(*
Nazwa:			P05_Weight
Opis:			Stacja wagi
Wersja:			v0.2
Data:			2019-10-1
Autor:			DP
Urzadzenia:		
Konfiguracja:	
Info:
-przerobione na wagę beckhofa
*)
PROGRAM P05_Weight
VAR_INPUT
	IbWeight1FormSensor						AT %I*		: BOOL;							//Czujnik nad Waga 1
	IbWeight2FormSensor						AT %I*		: BOOL;							//Czujnik nad Waga 2
	IbWeight3FormSensor						AT %I*		: BOOL;							//Czujnik nad Waga 3
	IbWeight4FormSensor						AT %I*		: BOOL;							//Czujnik nad Waga 4
	IbWeight5FormSensor						AT %I*		: BOOL;							//Czujnik nad Waga 4
	IbWeight6FormSensor						AT %I*		: BOOL;							//Czujnik nad Waga 4
END_VAR
VAR
	//Podnosnik szalek
	
	//eWeightLiftRunningState			:E_WeightLiftState;				// Stan pracy podajnika
	fbWeightLiftState					:FB_State;
	
	//Waga 1
	fbWeight1							:FB_BeckhoffEL3356Weight;		// Blok sterujący pierwszą wagą
	eWeight1State						:E_Station; 					// Stan pracy podajnika platynek			
	eWeight1RunningState				:E_WeightState; 				// Stan pracy podajnika platynek
	fbWeight1State						:FB_State;					

	(*No nowej wagi*)
	(*wejścia*)
	InWeight1Value						 AT %I*: DINT;			// Wartość wagi
	IbWeight1Overrange					 AT %I*: BOOL;						
	IbWeight1DataInvalid				 AT %I*: BOOL;		
	IbWeight1Error 						 AT %I*: BOOL;	
	IbWeight1CalibrationInProgress 		 AT %I*: BOOL;
	IbWeight1SteadyState				 AT %I*: BOOL;
	IbWeight1SyncError 					 AT %I*: BOOL;
	(*wyjścia*)
	QbWeight1StartCalibration 			 AT %Q*: BOOL;
	QbWeight1DisableCalibration     	 AT %Q*: BOOL;
	QbWeight1InputFreeze 				 AT %Q*: BOOL;
	QbWeight1SampleMode 				 AT %Q*: BOOL;
	QbWeight1Tara 					     AT %Q*: BOOL;
	
	(*Ostrzezenia*)
	bWeight1Warning1					:BOOL; // 
	tonWeight1Tare						:TON;
	
	//Waga 2
	fbWeight2							:FB_BeckhoffEL3356Weight;		// Blok sterujący pierwszą wagą
	eWeight2State						:E_Station; 					// Stan pracy podajnika platynek			
	eWeight2RunningState				:E_WeightState; 				// Stan pracy podajnika platynek
	fbWeight2State						:FB_State;					

	(*No nowej wagi*)
	(*wejścia*)
	InWeight2Value 						AT %I*: DINT;			// Wartość wagi
	IbWeight2Overrange 					AT %I*: BOOL;						
	IbWeight2DataInvalid 				AT %I*: BOOL;		
	IbWeight2Error 						AT %I*: BOOL;	
	IbWeight2CalibrationInProgress		AT %I*: BOOL;
	IbWeight2SteadyState 				AT %I*: BOOL;
	IbWeight2SyncError 					AT %I*: BOOL;
	(*wyjścia*)
	QbWeight2StartCalibration 			AT %Q*: BOOL;
	QbWeight2DisableCalibration			AT %Q*: BOOL;
	QbWeight2InputFreeze 				AT %Q*: BOOL;
	QbWeight2SampleMode 				AT %Q*: BOOL;
	QbWeight2Tara 						AT %Q*: BOOL;
	
	(*Ostrzezenia*)
	bWeight2Warning1					:BOOL; // 
	tonWeight2Tare						:TON;
		
	//Waga 3
	fbWeight3							:FB_BeckhoffEL3356Weight;		// Blok sterujący pierwszą wagą
	eWeight3State						:E_Station; 					// Stan pracy podajnika platynek			
	eWeight3RunningState				:E_WeightState; 				// Stan pracy podajnika platynek
	fbWeight3State						:FB_State;					

	(*No nowej wagi*)
	(*wejścia*)
	InWeight3Value						 AT %I*: DINT;			// Wartość wagi
	IbWeight3Overrange 					 AT %I*: BOOL;						
	IbWeight3DataInvalid 				 AT %I*: BOOL;		
	IbWeight3Error 						 AT %I*: BOOL;	
	IbWeight3CalibrationInProgress 		 AT %I*: BOOL;
	IbWeight3SteadyState 				 AT %I*: BOOL;
	IbWeight3SyncError 					 AT %I*: BOOL;
	(*wyjścia*)
	QbWeight3StartCalibration 			 AT %Q*: BOOL;
	QbWeight3DisableCalibration 		 AT %Q*: BOOL;
	QbWeight3InputFreeze 				 AT %Q*: BOOL;
	QbWeight3SampleMode 			   	 AT %Q*: BOOL;
	QbWeight3Tara 						 AT %Q*: BOOL;
	
	(*Ostrzezenia*)
	bWeight3Warning1					:BOOL; // 
	tonWeight3Tare						: TON;	
	
	//Waga 4
	fbWeight4							:FB_BeckhoffEL3356Weight;		// Blok sterujący pierwszą wagą
	eWeight4State						:E_Station; 					// Stan pracy podajnika platynek			
	eWeight4RunningState				:E_WeightState; 				// Stan pracy podajnika platynek
	fbWeight4State						:FB_State;					

	(*No nowej wagi*)
	(*wejścia*)
	InWeight4Value 						AT %I*: DINT;			// Wartość wagi
	IbWeight4Overrange 					AT %I*: BOOL;						
	IbWeight4DataInvalid				AT %I*: BOOL;		
	IbWeight4Error 						AT %I*: BOOL;	
	IbWeight4CalibrationInProgress 		AT %I*: BOOL;
	IbWeight4SteadyState 				AT %I*: BOOL;
	IbWeight4SyncError 					AT %I*: BOOL;
	(*wyjścia*)
	QbWeight4StartCalibration 			AT %Q*: BOOL;
	QbWeight4DisableCalibration 		AT %Q*: BOOL;
	QbWeight4InputFreeze 				AT %Q*: BOOL;
	QbWeight4SampleMode 				AT %Q*: BOOL;
	QbWeight4Tara 						AT %Q*: BOOL;

	(*Ostrzezenia*)
	bWeight4Warning1					:BOOL; // 
	tonWeight4Tare						:TON;	
		
(******** Dozowanie dwufazowe******)	
////// Wagi przy dozowaniu dwufazowym dodano 07.04.2022
	//Waga 5
	fbWeight5							:FB_BeckhoffEL3356Weight;		// Blok sterujący pierwszą wagą
	eWeight5State						:E_Station; 					// Stan pracy podajnika platynek			
	eWeight5RunningState				:E_WeightState; 				// Stan pracy podajnika platynek
	fbWeight5State						:FB_State;					

	(*No nowej wagi*)
	(*wejścia*)
	InWeight5Value 						AT %I*: DINT;			// Wartość wagi
	IbWeight5Overrange 					AT %I*: BOOL;						
	IbWeight5DataInvalid 				AT %I*: BOOL;		
	IbWeight5Error 						AT %I*: BOOL;	
	IbWeight5CalibrationInProgress 		AT %I*: BOOL;
	IbWeight5SteadyState 				AT %I*: BOOL;
	IbWeight5SyncError 					AT %I*: BOOL;
	(*wyjścia*)
	QbWeight5StartCalibration 			AT %Q*: BOOL;
	QbWeight5DisableCalibration 		AT %Q*: BOOL;
	QbWeight5InputFreeze 				AT %Q*: BOOL;
	QbWeight5SampleMode 				AT %Q*: BOOL;
	QbWeight5Tara 						AT %Q*: BOOL;

	(*Ostrzezenia*)
	bWeight5Warning1					:BOOL; // 
	tonWeight5Tare						:TON;		
	
	//Waga 5
	fbWeight6							:FB_BeckhoffEL3356Weight;		// Blok sterujący pierwszą wagą
	eWeight6State						:E_Station; 					// Stan pracy podajnika platynek			
	eWeight6RunningState				:E_WeightState; 				// Stan pracy podajnika platynek
	fbWeight6State						:FB_State;					

	(*No nowej wagi*)
	(*wejścia*)
	InWeight6Value 						AT %I*: DINT;			// Wartość wagi
	IbWeight6Overrange 					AT %I*: BOOL;						
	IbWeight6DataInvalid 				AT %I*: BOOL;		
	IbWeight6Error 						AT %I*: BOOL;	
	IbWeight6CalibrationInProgress 		AT %I*: BOOL;
	IbWeight6SteadyState 				AT %I*: BOOL;
	IbWeight6SyncError 					AT %I*: BOOL;
	(*wyjścia*)
	QbWeight6StartCalibration 			AT %Q*: BOOL;
	QbWeight6DisableCalibration 		AT %Q*: BOOL;
	QbWeight6InputFreeze 				AT %Q*: BOOL;
	QbWeight6SampleMode 				AT %Q*: BOOL;
	QbWeight6Tara 						AT %Q*: BOOL;

	(*Ostrzezenia*)
	bWeight6Warning1					:BOOL; // 
	tonWeight6Tare						:TON;		
	
(******** Dozowanie dwufazowe******)		
	
	//Czujniki optyczne przed i za wagą
	fbFilterWeight1: FB_FilterEx;
	fbFilterWeight2: FB_FilterEx;
	fbFilterWeight3: FB_FilterEx;
	fbFilterWeight4: FB_FilterEx;
	fbFilterWeight5: FB_FilterEx;(****** dodane 07.04.2022 przy dodzowniu dwufazowym	**)
	fbFilterWeight6: FB_FilterEx;(****** dodane 07.04.2022 przy dodzowniu dwufazowym	**)

	rFilteredWeight1Value: REAL;
	rFilteredWeight2Value: REAL;
	rFilteredWeight3Value: REAL;
	rFilteredWeight4Value: REAL;
	rFilteredWeight5Value: REAL;(****** dodane 07.04.2022 przy dodzowniu dwufazowym	**)
	rFilteredWeight6Value: REAL;(****** dodane 07.04.2022 przy dodzowniu dwufazowym	**)
	
	//Damian dodane 2 fazy
	fbWeightStation2Phase							: FB_WeightStation;	
	eWeightStation2PhaseState						: E_Station;
	eWeightStation2PhaseRunningState				: E_WeightLiftStationState;
	
	//Dodane Przez Mikołaja
	fbWeightStation									: FB_WeightStation;
	eWeightStationState								: E_Station;
	eWeightStationRunningState						: E_WeightLiftStationState;
	
	IbWeight1ActuatorSensorUp			AT %I*		: BOOL;							//Czujnik podnoszenia Waga 1
	IbWeight2ActuatorSensorUp			AT %I*		: BOOL;							//Czujnik podnoszenia Waga 2
	IbWeight3ActuatorSensorUp			AT %I*		: BOOL;							//Czujnik podnoszenia Waga 3
	IbWeight4ActuatorSensorUp			AT %I*		: BOOL;							//Czujnik podnoszenia Waga 4
	IbWeight5ActuatorSensorUp			AT %I*		: BOOL;							//Czujnik podnoszenia Waga 5 
	IbWeight6ActuatorSensorUp			AT %I*		: BOOL;							//Czujnik podnoszenia Waga 6 
		
	QbWeight1Actuator								: BOOL;							//Podnoszenie Waga 1
    QbWeight2Actuator								: BOOL;							//Podnoszenie Waga 2
	QbWeight3Actuator								: BOOL;							//Podnoszenie Waga 3
	QbWeight4Actuator								: BOOL;							//Podnoszenie Waga 4	                                    		
	QbWeight5Actuator								: BOOL;							//Podnoszenie Waga 5 (2faza)	                                    		
	QbWeight6Actuator								: BOOL;							//Podnoszenie Waga 6 (2faza)

		
	(*Symulacja czujników*)
	tonIbWeight1ActuatorSensorUp					: TON;	
	tonIbWeight2ActuatorSensorUp					: TON;	
	tonIbWeight3ActuatorSensorUp					: TON;	
	tonIbWeight4ActuatorSensorUp					: TON;	
	tonIbWeight5ActuatorSensorUp					: TON;	
	tonIbWeight6ActuatorSensorUp					: TON;	
	
	tonIbWeight1FormSensor: TON;
	tonIbWeight2FormSensor: TON;
	tonIbWeight3FormSensor: TON;
	tonIbWeight4FormSensor: TON;
	tonIbWeight5FormSensor: TON;
	tonIbWeight6FormSensor: TON;
	
	fbIbWeight1FormBeforeSensor: FB_InputFilter_v2;
	fbIbWeight2FormBeforeSensor: FB_InputFilter_v2;
	fbIbWeight3FormBeforeSensor: FB_InputFilter_v2;
	fbIbWeight4FormBeforeSensor: FB_InputFilter_v2;		
	fbIbWeight5FormBeforeSensor: FB_InputFilter_v2;		
	fbIbWeight6FormBeforeSensor: FB_InputFilter_v2;			
	btemp: BOOL;
	
	//wykresy
	fbTrig1 : R_TRIG;
    fbTrig2 : R_TRIG;
    fbTrig3 : R_TRIG;
    fbTrig4 : R_TRIG;
	tSys : DT;
    tTOD : TOD;
	GetTimeSeconds : INT;
	weightIndex : INT;   // 0..7
    valueY : INT;
	i : INT;
	 
	fbHistory: FB_WeightHistory;
END_VAR


fbWeight1.bIgnoreError:=fbWeight2.bIgnoreError:=fbWeight3.bIgnoreError:=fbWeight4.bIgnoreError:=fbWeight5.bIgnoreError:=fbWeight6.bIgnoreError;

aFilter();
aWeight1();
aWeight2();
aWeight3();
aWeight4();
aWeight5();
aWeight6();
ACT_WeightChartDrawers();
IF NOT bDosingTwoPhases THEN
	ACT_WeightStation();
ELSE
	ACT_WeightStation2Phase();
END_IF

// Czas opóżnienia zbierania próbekFB_EntranceGatesServo
fbWeight1.nWeightingDelay:=fbWeight2.nWeightingDelay:=fbWeight3.nWeightingDelay:=fbWeight4.nWeightingDelay:=530;//530
fbWeight5.nWeightingDelay:=fbWeight6.nWeightingDelay:=750;//było 685

(********* GENEROWANIE STANU STACJI DO WIZKI**********)

fbWeight1State(
	eState															:= eWeight1State , 
	bRun															:= VIS.bWeight1DoWeighting,	
	eWeightRunningState												:= eWeight1RunningState , 
	sStateDesc														=> VIS.sWeight1State,
	iState															=> VIS.iWeight1State	);	

fbWeight2State(
	eState															:= eWeight2State , 
	bRun															:= VIS.bWeight2DoWeighting,	
	eWeightRunningState												:= eWeight2RunningState , 
	sStateDesc														=> VIS.sWeight2State,
	iState															=> VIS.iWeight2State	);	
		
fbWeight3State(
	eState															:= eWeight3State , 
	bRun															:= VIS.bWeight3DoWeighting,	
	eWeightRunningState												:= eWeight3RunningState , 
	sStateDesc														=> VIS.sWeight3State,
	iState															=> VIS.iWeight3State	);	
	
fbWeight4State(
	eState															:= eWeight4State , 
	bRun															:= VIS.bWeight4DoWeighting,	
	eWeightRunningState												:= eWeight4RunningState , 
	sStateDesc														=> VIS.sWeight4State,
	iState															=> VIS.iWeight4State	);	
	
fbWeight5State(
	eState															:= eWeight5State , 
	bRun															:= VIS.bWeight5DoWeighting,	
	eWeightRunningState												:= eWeight5RunningState , 
	sStateDesc														=> VIS.sWeight5State,
	iState															=> VIS.iWeight5State	);	

fbWeight6State(
	eState															:= eWeight6State , 
	bRun															:= VIS.bWeight6DoWeighting,	
	eWeightRunningState												:= eWeight6RunningState , 
	sStateDesc														=> VIS.sWeight6State,
	iState															=> VIS.iWeight6State	);		
	
fbWeightLiftState(
	eState															:= eWeightStationState, 
	bRun															:= VIS.bWeightLiftRun OR bWeightLift2PhaseRun,	
	eWeightLiftRunningState											:= eWeightStationRunningState , 
	sStateDesc														=> VIS.sWeightLiftState,
	iState															=> VIS.iWeightLiftState	);		
	
(***** KONIEC GENEROWANIE STANU STACJI DO WIZKI*******)

(****Ostrzezenia***)
// Waga 1
WeightWarning[0].sDescription										:= 'Wagi | Brak stabilizacji przy pomiarach';
IF (bWeight1Warning1 OR bWeight2Warning1 OR bWeight3Warning1 OR bWeight4Warning1 OR bWeight5Warning1 OR bWeight6Warning1) AND NOT WeightWarning[0].bWarning THEN
	WeightWarning[0].bWarning										:= TRUE;
	
ELSIF NOT bWeight1Warning1 AND WeightWarning[0].bAcknowledge THEN
	WeightWarning[0].bWarning										:= FALSE;
	WeightWarning[0].bAcknowledge									:= FALSE;
	VIS.uliWarningAcknowledge.4 										:= FALSE;
	
ELSIF WeightWarning[0].bAcknowledge THEN
	WeightWarning[0].bAcknowledge									:= TRUE;
END_IF


(********KASOWANIE ROZKAZÓW CYKLI*********)
IF fbWeight1.bCycleDone AND bManualMode THEN
	VIS.bWeight1DoWeighting 												:= FALSE;
END_IF

tonWeight1Tare(IN:=VIS.bWeight1Tare,PT:=T#2S);
IF tonWeight1Tare.Q THEN
	VIS.bWeight1Tare												:= FALSE;
END_IF

IF fbWeight2.bCycleDone AND bManualMode THEN
	VIS.bWeight2DoWeighting 												:= FALSE;
END_IF

tonWeight2Tare(IN:=VIS.bWeight2Tare,PT:=T#2S);
IF tonWeight2Tare.Q THEN
	VIS.bWeight2Tare												:= FALSE;
END_IF

IF fbWeight3.bCycleDone AND bManualMode THEN
	VIS.bWeight3DoWeighting 												:= FALSE;
END_IF

tonWeight3Tare(IN:=VIS.bWeight3Tare,PT:=T#2S);
IF tonWeight3Tare.Q THEN
	VIS.bWeight3Tare												:= FALSE;
END_IF
//
IF fbWeight4.bCycleDone AND bManualMode THEN
	VIS.bWeight4DoWeighting 												:= FALSE;
END_IF

tonWeight4Tare(IN:=VIS.bWeight4Tare,PT:=T#2S);
IF tonWeight4Tare.Q THEN
	VIS.bWeight4Tare												:= FALSE;
END_IF

// Waga 5 (1 stacja przy dwufazie)
IF fbWeight5.bCycleDone AND bManualMode THEN
	VIS.bWeight5DoWeighting 												:= FALSE;
END_IF

tonWeight5Tare(IN:=VIS.bWeight5Tare,PT:=T#2S);
IF tonWeight5Tare.Q THEN
	VIS.bWeight5Tare												:= FALSE;
END_IF

// Waga 6 (1 stacja przy dwufazie)
IF fbWeight6.bCycleDone AND bManualMode THEN
	VIS.bWeight6DoWeighting 												:= FALSE;
END_IF

tonWeight6Tare(IN:=VIS.bWeight6Tare,PT:=T#2S);
IF tonWeight6Tare.Q THEN
	VIS.bWeight6Tare												:= FALSE;
END_IF
(*****KONIEC KASOWANIA ROZKAZÓW CYKLI*****)

(**SYMULACJA CZUJNIKÓW**)
tonIbWeight1ActuatorSensorUp(IN:= QbWeight1Actuator, PT:=T#80MS);
tonIbWeight2ActuatorSensorUp(IN:= QbWeight2Actuator, PT:=T#80MS);
tonIbWeight3ActuatorSensorUp(IN:= QbWeight3Actuator, PT:=T#80MS);
tonIbWeight4ActuatorSensorUp(IN:= QbWeight4Actuator, PT:=T#80MS);
tonIbWeight5ActuatorSensorUp(IN:= QbWeight5Actuator, PT:=T#100MS);
tonIbWeight6ActuatorSensorUp(IN:= QbWeight6Actuator, PT:=T#100MS);

ACTION ACT_WeightChartDrawers:
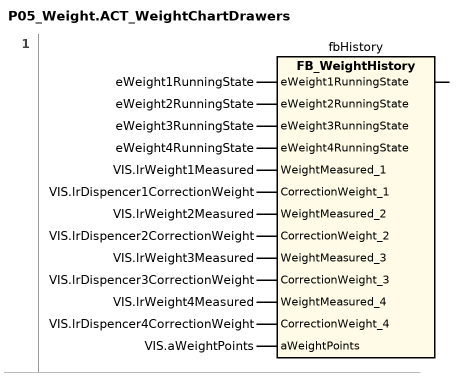
// NETWORK 1
fbHistory(
    eWeight1RunningState := eWeight1RunningState,
    eWeight2RunningState := eWeight2RunningState,
    eWeight3RunningState := eWeight3RunningState,
    eWeight4RunningState := eWeight4RunningState,
    WeightMeasured_1 := VIS.lrWeight1Measured,
    CorrectionWeight_1 := VIS.lrDispencer1CorrectionWeight,
    WeightMeasured_2 := VIS.lrWeight2Measured,
    CorrectionWeight_2 := VIS.lrDispencer2CorrectionWeight,
    WeightMeasured_3 := VIS.lrWeight3Measured,
    CorrectionWeight_3 := VIS.lrDispencer3CorrectionWeight,
    WeightMeasured_4 := VIS.lrWeight4Measured,
    CorrectionWeight_4 := VIS.lrDispencer4CorrectionWeight,
    aWeightPoints := VIS.aWeightPoints); // FB_WeightHistory
END_ACTION

ACTION ACT_WeightStation:
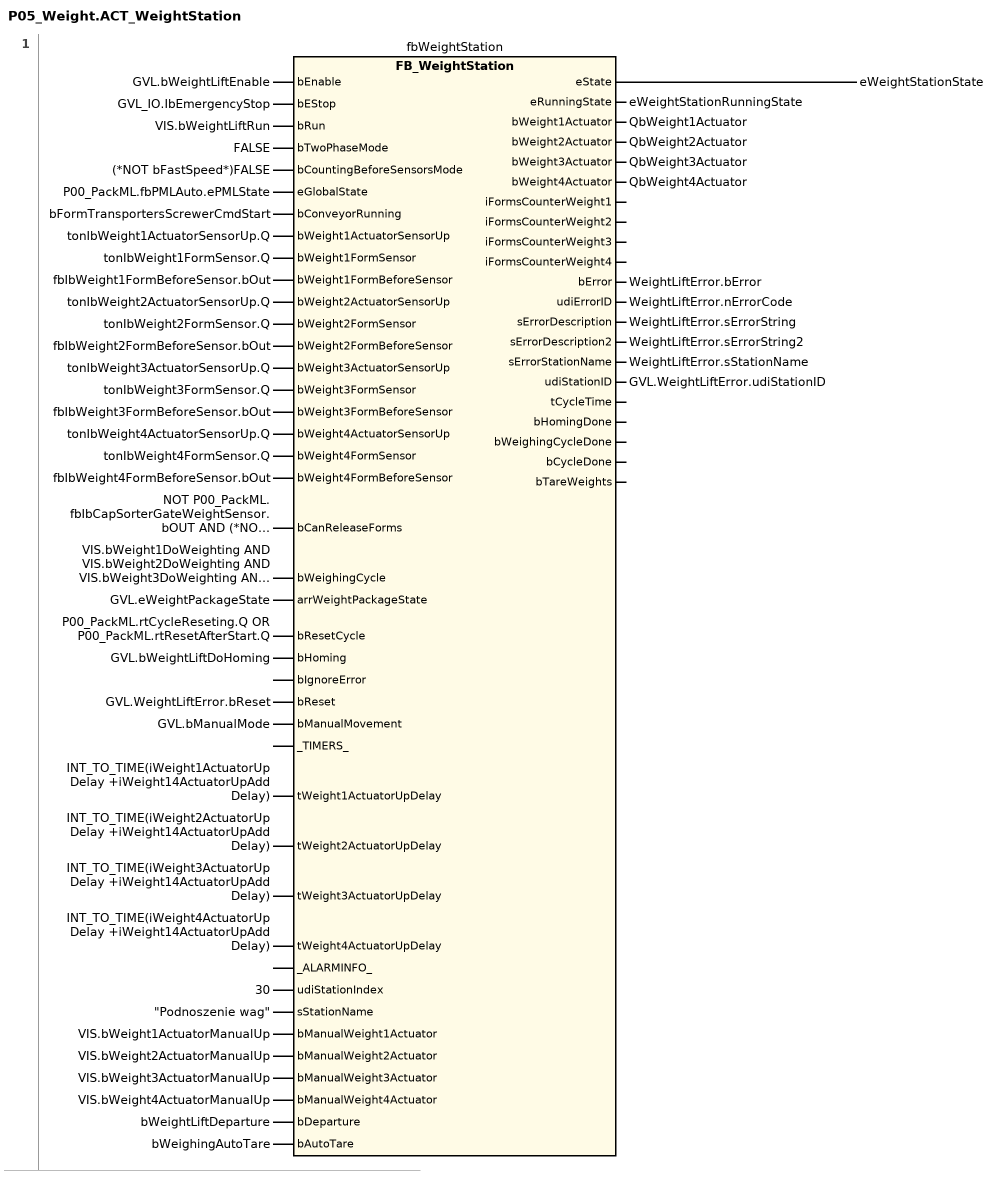
// NETWORK 1
fbWeightStation(
    bEnable := GVL.bWeightLiftEnable,
    bEStop := GVL_IO.IbEmergencyStop,
    bRun := VIS.bWeightLiftRun,
    bTwoPhaseMode := FALSE,
    bCountingBeforeSensorsMode := (*NOT bFastSpeed*)FALSE,
    eGlobalState := P00_PackML.fbPMLAuto.ePMLState,
    bConveyorRunning := bFormTransportersScrewerCmdStart,
    bWeight1ActuatorSensorUp := tonIbWeight1ActuatorSensorUp.Q,
    bWeight1FormSensor := tonIbWeight1FormSensor.Q,
    bWeight1FormBeforeSensor := fbIbWeight1FormBeforeSensor.bOut,
    bWeight2ActuatorSensorUp := tonIbWeight2ActuatorSensorUp.Q,
    bWeight2FormSensor := tonIbWeight2FormSensor.Q,
    bWeight2FormBeforeSensor := fbIbWeight2FormBeforeSensor.bOut,
    bWeight3ActuatorSensorUp := tonIbWeight3ActuatorSensorUp.Q,
    bWeight3FormSensor := tonIbWeight3FormSensor.Q,
    bWeight3FormBeforeSensor := fbIbWeight3FormBeforeSensor.bOut,
    bWeight4ActuatorSensorUp := tonIbWeight4ActuatorSensorUp.Q,
    bWeight4FormSensor := tonIbWeight4FormSensor.Q,
    bWeight4FormBeforeSensor := fbIbWeight4FormBeforeSensor.bOut,
    bCanReleaseForms := NOT P00_PackML.fbIbCapSorterGateWeightSensor.bOUT AND (*NOT P00_PackML.fbIbCapCorrectCheckFormSensor.bOUT AND zalezy od ilosci formatek*)  NOT bWeight1234ReleaseBlock,
    bWeighingCycle := VIS.bWeight1DoWeighting AND VIS.bWeight2DoWeighting AND VIS.bWeight3DoWeighting AND VIS.bWeight4DoWeighting,
    arrWeightPackageState := GVL.eWeightPackageState,
    bResetCycle := P00_PackML.rtCycleReseting.Q OR P00_PackML.rtResetAfterStart.Q,
    bHoming := GVL.bWeightLiftDoHoming,
    bReset := GVL.WeightLiftError.bReset,
    bManualMovement := GVL.bManualMode,
    tWeight1ActuatorUpDelay := INT_TO_TIME(iWeight1ActuatorUpDelay +iWeight14ActuatorUpAddDelay),
    tWeight2ActuatorUpDelay := INT_TO_TIME(iWeight2ActuatorUpDelay +iWeight14ActuatorUpAddDelay),
    tWeight3ActuatorUpDelay := INT_TO_TIME(iWeight3ActuatorUpDelay +iWeight14ActuatorUpAddDelay),
    tWeight4ActuatorUpDelay := INT_TO_TIME(iWeight4ActuatorUpDelay +iWeight14ActuatorUpAddDelay),
    udiStationIndex := 30,
    sStationName := "Podnoszenie wag",
    bManualWeight1Actuator := VIS.bWeight1ActuatorManualUp,
    bManualWeight2Actuator := VIS.bWeight2ActuatorManualUp,
    bManualWeight3Actuator := VIS.bWeight3ActuatorManualUp,
    bManualWeight4Actuator := VIS.bWeight4ActuatorManualUp,
    bDeparture := bWeightLiftDeparture,
    bAutoTare := bWeighingAutoTare,
    eRunningState => eWeightStationRunningState,
    bWeight1Actuator => QbWeight1Actuator,
    bWeight2Actuator => QbWeight2Actuator,
    bWeight3Actuator => QbWeight3Actuator,
    bWeight4Actuator => QbWeight4Actuator,
    bError => WeightLiftError.bError,
    udiErrorID => WeightLiftError.nErrorCode,
    sErrorDescription => WeightLiftError.sErrorString,
    sErrorDescription2 => WeightLiftError.sErrorString2,
    sErrorStationName => WeightLiftError.sStationName,
    udiStationID => GVL.WeightLiftError.udiStationID); // FB_WeightStation
eWeightStationState := fbWeightStation.eState;
END_ACTION

ACTION ACT_WeightStation2Phase:
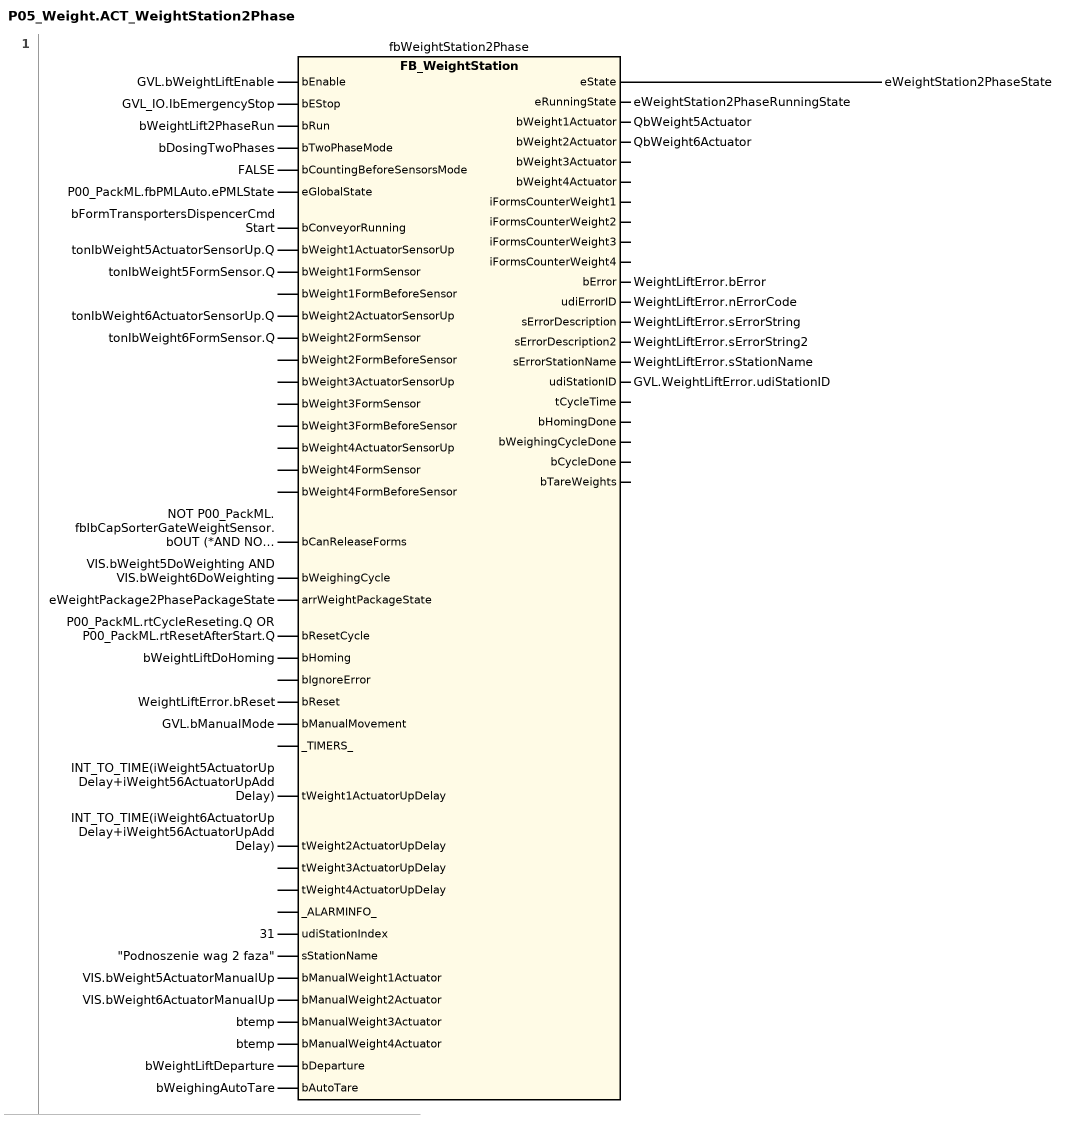
// NETWORK 1
fbWeightStation2Phase(
    bEnable := GVL.bWeightLiftEnable,
    bEStop := GVL_IO.IbEmergencyStop,
    bRun := bWeightLift2PhaseRun,
    bTwoPhaseMode := bDosingTwoPhases,
    bCountingBeforeSensorsMode := FALSE,
    eGlobalState := P00_PackML.fbPMLAuto.ePMLState,
    bConveyorRunning := bFormTransportersDispencerCmdStart,
    bWeight1ActuatorSensorUp := tonIbWeight5ActuatorSensorUp.Q,
    bWeight1FormSensor := tonIbWeight5FormSensor.Q,
    bWeight2ActuatorSensorUp := tonIbWeight6ActuatorSensorUp.Q,
    bWeight2FormSensor := tonIbWeight6FormSensor.Q,
    bCanReleaseForms := NOT P00_PackML.fbIbCapSorterGateWeightSensor.bOUT (*AND NOT P00_PackML.fbIbCapCorrectCheckFormSensor.bOUT*)  AND NOT bWeight56ReleaseBlock,
    bWeighingCycle := VIS.bWeight5DoWeighting AND VIS.bWeight6DoWeighting,
    arrWeightPackageState := eWeightPackage2PhasePackageState,
    bResetCycle := P00_PackML.rtCycleReseting.Q OR P00_PackML.rtResetAfterStart.Q,
    bHoming := bWeightLiftDoHoming,
    bReset := WeightLiftError.bReset,
    bManualMovement := GVL.bManualMode,
    tWeight1ActuatorUpDelay := INT_TO_TIME(iWeight5ActuatorUpDelay+iWeight56ActuatorUpAddDelay),
    tWeight2ActuatorUpDelay := INT_TO_TIME(iWeight6ActuatorUpDelay+iWeight56ActuatorUpAddDelay),
    udiStationIndex := 31,
    sStationName := "Podnoszenie wag 2 faza",
    bManualWeight1Actuator := VIS.bWeight5ActuatorManualUp,
    bManualWeight2Actuator := VIS.bWeight6ActuatorManualUp,
    bManualWeight3Actuator := btemp,
    bManualWeight4Actuator := btemp,
    bDeparture := bWeightLiftDeparture,
    bAutoTare := bWeighingAutoTare,
    eRunningState => eWeightStation2PhaseRunningState,
    bWeight1Actuator => QbWeight5Actuator,
    bWeight2Actuator => QbWeight6Actuator,
    bError => WeightLiftError.bError,
    udiErrorID => WeightLiftError.nErrorCode,
    sErrorDescription => WeightLiftError.sErrorString,
    sErrorDescription2 => WeightLiftError.sErrorString2,
    sErrorStationName => WeightLiftError.sStationName,
    udiStationID => GVL.WeightLiftError.udiStationID); // FB_WeightStation
eWeightStation2PhaseState := fbWeightStation2Phase.eState;
END_ACTION

ACTION aFilter:
fbFilterWeight1(
				rIn:=				DINT_TO_REAL(InWeight1Value), 
				tTimeConstant:= 	T#25MS, //bylo 25
				rOut=>				rFilteredWeight1Value);
							
fbFilterWeight2(
				rIn:=				DINT_TO_REAL(InWeight2Value), 
				tTimeConstant:= 	T#25MS, //bylo 25
				rOut=>				rFilteredWeight2Value);
				
fbFilterWeight3(
				rIn:=				DINT_TO_REAL(InWeight3Value), 
				tTimeConstant:= 	T#52MS, //bylo 25
				rOut=>				rFilteredWeight3Value);
				
fbFilterWeight4(
				rIn:=				DINT_TO_REAL(InWeight4Value), 
				tTimeConstant:= 	T#25MS, //bylo 25
				rOut=>				rFilteredWeight4Value);
///////////////////////////////////////////////////////////////////////////////				
fbFilterWeight5(
				rIn:=				DINT_TO_REAL(InWeight5Value), 
				tTimeConstant:= 	T#25MS, //bylo 25
				rOut=>				rFilteredWeight5Value);
								
fbFilterWeight6(
				rIn:=				DINT_TO_REAL(InWeight6Value), 
				tTimeConstant:= 	T#25MS, //bylo 25
				rOut=>				rFilteredWeight6Value);														
/////////////////////////////////////////////////////////////////////////////

tonIbWeight1FormSensor			(IN:=IbWeight1FormSensor ,		PT:=T#120MS); //160
tonIbWeight2FormSensor			(IN:=IbWeight2FormSensor ,		PT:=T#120MS); //160
tonIbWeight3FormSensor			(IN:=IbWeight3FormSensor ,		PT:=T#120MS); //160
tonIbWeight4FormSensor			(IN:=IbWeight4FormSensor ,		PT:=T#120MS); //160
tonIbWeight5FormSensor			(IN:=IbWeight5FormSensor ,		PT:=T#120MS); //60
tonIbWeight6FormSensor			(IN:=IbWeight6FormSensor ,		PT:=T#120MS); //60

IF VIS.nFormTransportersScrewerVelocitySVShow < 500 THEN
	fbIbWeight1FormBeforeSensor	(bIN:=IbWeight1ActuatorSensorUp,	tFilterTimeOn:=T#70MS,	tFilterTimeOff:=T#150MS);
	fbIbWeight2FormBeforeSensor	(bIN:=IbWeight2ActuatorSensorUp,	tFilterTimeOn:=T#70MS,	tFilterTimeOff:=T#150MS);
	fbIbWeight3FormBeforeSensor	(bIN:=IbWeight3ActuatorSensorUp,	tFilterTimeOn:=T#70MS,	tFilterTimeOff:=T#150MS);
	fbIbWeight4FormBeforeSensor	(bIN:=IbWeight4ActuatorSensorUp,	tFilterTimeOn:=T#70MS,	tFilterTimeOff:=T#150MS);
ELSE
	fbIbWeight1FormBeforeSensor	(bIN:=IbWeight1ActuatorSensorUp,	tFilterTimeOn:=T#10MS,	tFilterTimeOff:=T#10MS);//bylo 40 i 20
	fbIbWeight2FormBeforeSensor	(bIN:=IbWeight2ActuatorSensorUp,	tFilterTimeOn:=T#10MS,	tFilterTimeOff:=T#10MS);//bylo 40 i 20
	fbIbWeight3FormBeforeSensor	(bIN:=IbWeight3ActuatorSensorUp,	tFilterTimeOn:=T#10MS,	tFilterTimeOff:=T#10MS);//bylo 40 i 20
	fbIbWeight4FormBeforeSensor	(bIN:=IbWeight4ActuatorSensorUp,	tFilterTimeOn:=T#10MS,	tFilterTimeOff:=T#10MS);//bylo 40 i 20	
END_IF

IF VIS.nFormTransportersDispencerVelocitySVShow < 500 THEN
	fbIbWeight5FormBeforeSensor	(bIN:=IbWeight5FormSensor,			tFilterTimeOn:=T#70MS,	tFilterTimeOff:=T#150MS);
	fbIbWeight6FormBeforeSensor	(bIN:=IbWeight6FormSensor,			tFilterTimeOn:=T#70MS,	tFilterTimeOff:=T#150MS);
ELSE
	fbIbWeight5FormBeforeSensor	(bIN:=IbWeight5FormSensor,			tFilterTimeOn:=T#70MS,	tFilterTimeOff:=T#150MS);
	fbIbWeight6FormBeforeSensor	(bIN:=IbWeight6FormSensor,			tFilterTimeOn:=T#70MS,	tFilterTimeOff:=T#150MS);
END_IF
END_ACTION

ACTION aWeight1:
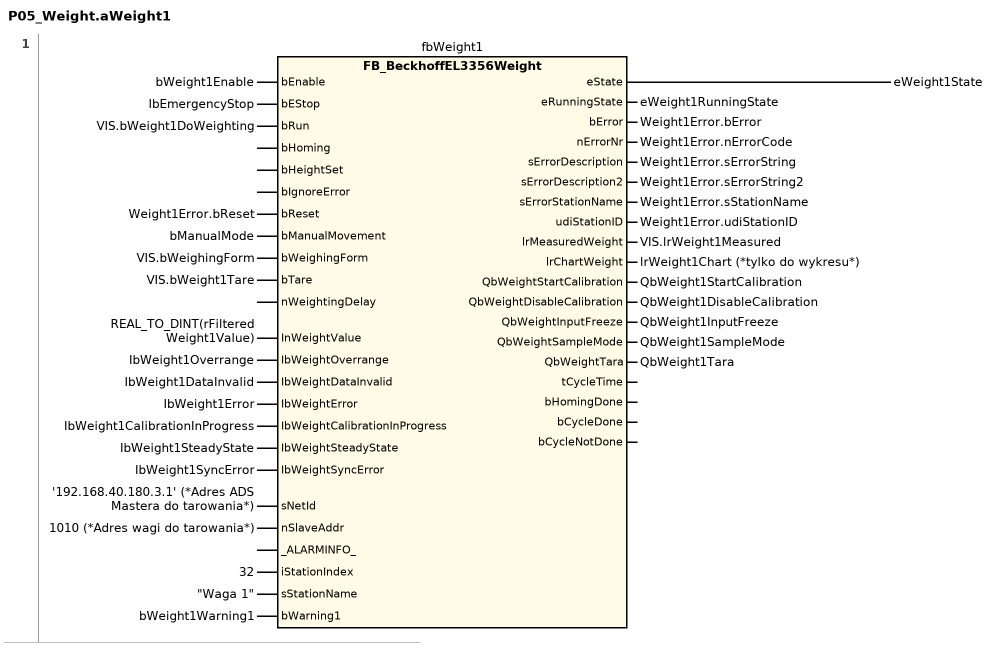
// NETWORK 1
fbWeight1(
    bEnable := bWeight1Enable,
    bEStop := IbEmergencyStop,
    bRun := VIS.bWeight1DoWeighting,
    bReset := Weight1Error.bReset,
    bManualMovement := bManualMode,
    bWeighingForm := VIS.bWeighingForm,
    bTare := VIS.bWeight1Tare,
    InWeightValue := REAL_TO_DINT(rFilteredWeight1Value),
    IbWeightOverrange := IbWeight1Overrange,
    IbWeightDataInvalid := IbWeight1DataInvalid,
    IbWeightError := IbWeight1Error,
    IbWeightCalibrationInProgress := IbWeight1CalibrationInProgress,
    IbWeightSteadyState := IbWeight1SteadyState,
    IbWeightSyncError := IbWeight1SyncError,
    sNetId := '192.168.40.180.3.1' (*Adres ADS Mastera do tarowania*),
    nSlaveAddr := 1010 (*Adres wagi do tarowania*),
    iStationIndex := 32,
    sStationName := "Waga 1",
    bWarning1 := bWeight1Warning1,
    eRunningState => eWeight1RunningState,
    bError => Weight1Error.bError,
    nErrorNr => Weight1Error.nErrorCode,
    sErrorDescription => Weight1Error.sErrorString,
    sErrorDescription2 => Weight1Error.sErrorString2,
    sErrorStationName => Weight1Error.sStationName,
    udiStationID => Weight1Error.udiStationID,
    lrMeasuredWeight => VIS.lrWeight1Measured,
    lrChartWeight => lrWeight1Chart (*tylko do wykresu*),
    QbWeightStartCalibration => QbWeight1StartCalibration,
    QbWeightDisableCalibration => QbWeight1DisableCalibration,
    QbWeightInputFreeze => QbWeight1InputFreeze,
    QbWeightSampleMode => QbWeight1SampleMode,
    QbWeightTara => QbWeight1Tara); // FB_BeckhoffEL3356Weight
eWeight1State := fbWeight1.eState;
END_ACTION

ACTION aWeight2:
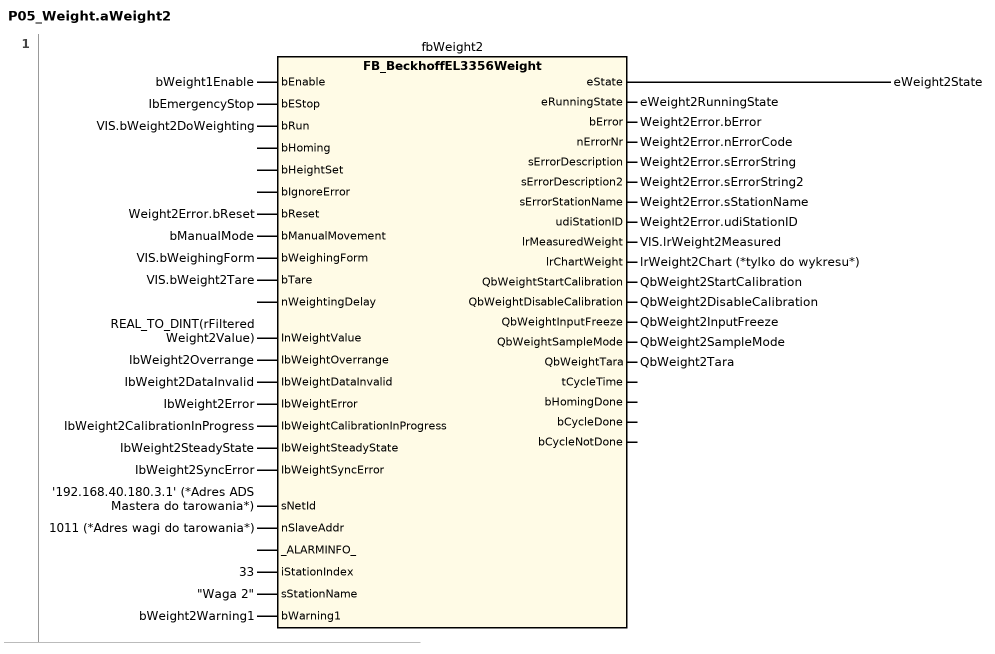
// NETWORK 1
fbWeight2(
    bEnable := bWeight1Enable,
    bEStop := IbEmergencyStop,
    bRun := VIS.bWeight2DoWeighting,
    bReset := Weight2Error.bReset,
    bManualMovement := bManualMode,
    bWeighingForm := VIS.bWeighingForm,
    bTare := VIS.bWeight2Tare,
    InWeightValue := REAL_TO_DINT(rFilteredWeight2Value),
    IbWeightOverrange := IbWeight2Overrange,
    IbWeightDataInvalid := IbWeight2DataInvalid,
    IbWeightError := IbWeight2Error,
    IbWeightCalibrationInProgress := IbWeight2CalibrationInProgress,
    IbWeightSteadyState := IbWeight2SteadyState,
    IbWeightSyncError := IbWeight2SyncError,
    sNetId := '192.168.40.180.3.1' (*Adres ADS Mastera do tarowania*),
    nSlaveAddr := 1011 (*Adres wagi do tarowania*),
    iStationIndex := 33,
    sStationName := "Waga 2",
    bWarning1 := bWeight2Warning1,
    eRunningState => eWeight2RunningState,
    bError => Weight2Error.bError,
    nErrorNr => Weight2Error.nErrorCode,
    sErrorDescription => Weight2Error.sErrorString,
    sErrorDescription2 => Weight2Error.sErrorString2,
    sErrorStationName => Weight2Error.sStationName,
    udiStationID => Weight2Error.udiStationID,
    lrMeasuredWeight => VIS.lrWeight2Measured,
    lrChartWeight => lrWeight2Chart (*tylko do wykresu*),
    QbWeightStartCalibration => QbWeight2StartCalibration,
    QbWeightDisableCalibration => QbWeight2DisableCalibration,
    QbWeightInputFreeze => QbWeight2InputFreeze,
    QbWeightSampleMode => QbWeight2SampleMode,
    QbWeightTara => QbWeight2Tara); // FB_BeckhoffEL3356Weight
eWeight2State := fbWeight2.eState;
END_ACTION

ACTION aWeight3:
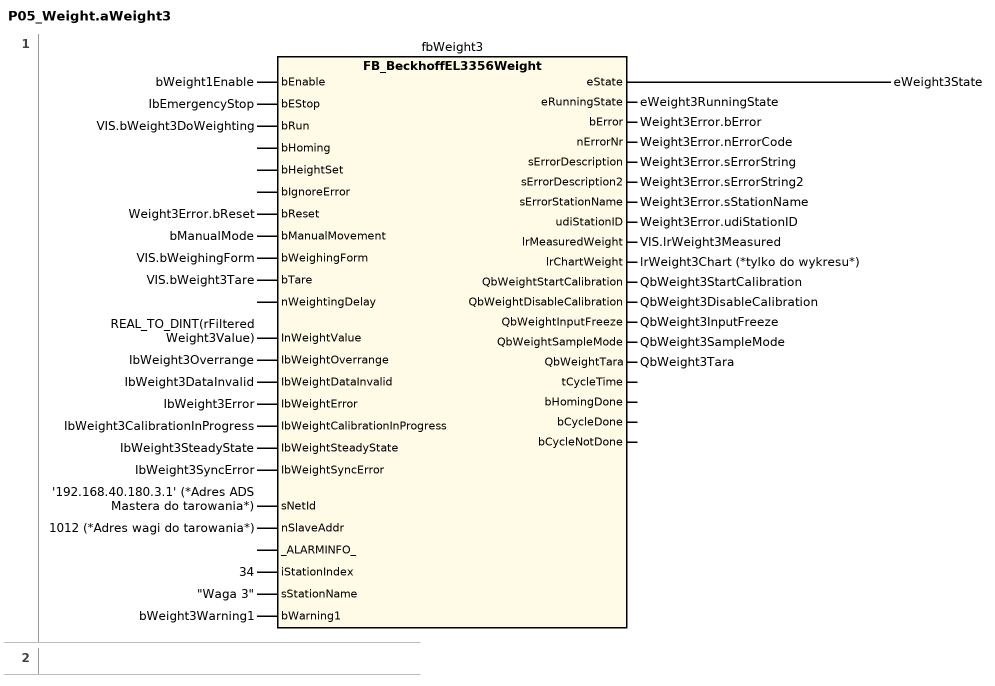
// NETWORK 1
fbWeight3(
    bEnable := bWeight1Enable,
    bEStop := IbEmergencyStop,
    bRun := VIS.bWeight3DoWeighting,
    bReset := Weight3Error.bReset,
    bManualMovement := bManualMode,
    bWeighingForm := VIS.bWeighingForm,
    bTare := VIS.bWeight3Tare,
    InWeightValue := REAL_TO_DINT(rFilteredWeight3Value),
    IbWeightOverrange := IbWeight3Overrange,
    IbWeightDataInvalid := IbWeight3DataInvalid,
    IbWeightError := IbWeight3Error,
    IbWeightCalibrationInProgress := IbWeight3CalibrationInProgress,
    IbWeightSteadyState := IbWeight3SteadyState,
    IbWeightSyncError := IbWeight3SyncError,
    sNetId := '192.168.40.180.3.1' (*Adres ADS Mastera do tarowania*),
    nSlaveAddr := 1012 (*Adres wagi do tarowania*),
    iStationIndex := 34,
    sStationName := "Waga 3",
    bWarning1 := bWeight3Warning1,
    eRunningState => eWeight3RunningState,
    bError => Weight3Error.bError,
    nErrorNr => Weight3Error.nErrorCode,
    sErrorDescription => Weight3Error.sErrorString,
    sErrorDescription2 => Weight3Error.sErrorString2,
    sErrorStationName => Weight3Error.sStationName,
    udiStationID => Weight3Error.udiStationID,
    lrMeasuredWeight => VIS.lrWeight3Measured,
    lrChartWeight => lrWeight3Chart (*tylko do wykresu*),
    QbWeightStartCalibration => QbWeight3StartCalibration,
    QbWeightDisableCalibration => QbWeight3DisableCalibration,
    QbWeightInputFreeze => QbWeight3InputFreeze,
    QbWeightSampleMode => QbWeight3SampleMode,
    QbWeightTara => QbWeight3Tara); // FB_BeckhoffEL3356Weight
eWeight3State := fbWeight3.eState;

// NETWORK 2
END_ACTION

ACTION aWeight4:
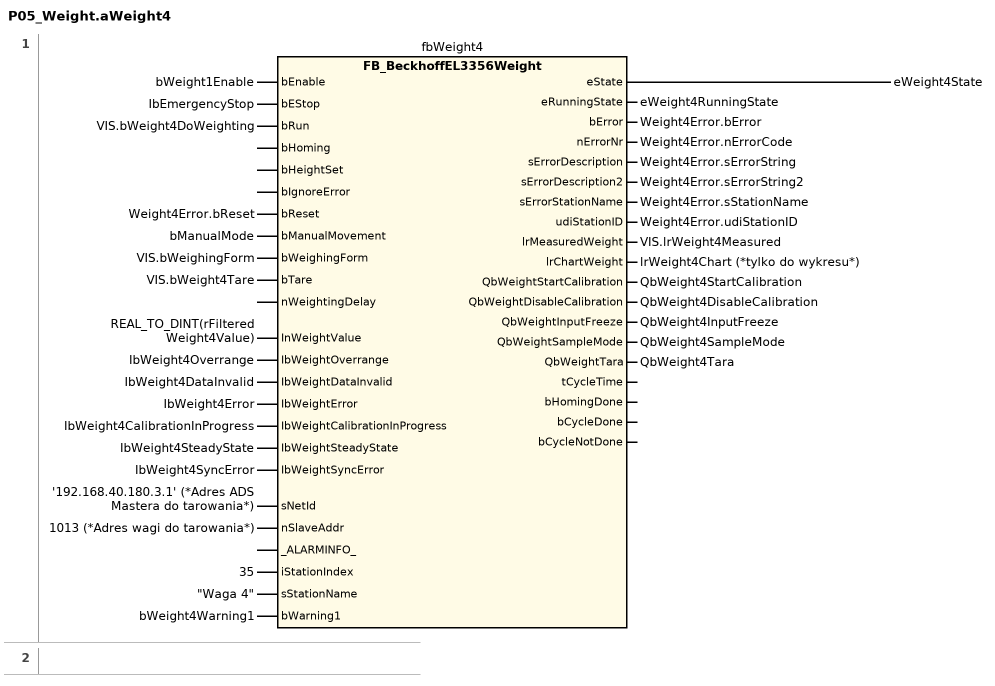
// NETWORK 1
fbWeight4(
    bEnable := bWeight1Enable,
    bEStop := IbEmergencyStop,
    bRun := VIS.bWeight4DoWeighting,
    bReset := Weight4Error.bReset,
    bManualMovement := bManualMode,
    bWeighingForm := VIS.bWeighingForm,
    bTare := VIS.bWeight4Tare,
    InWeightValue := REAL_TO_DINT(rFilteredWeight4Value),
    IbWeightOverrange := IbWeight4Overrange,
    IbWeightDataInvalid := IbWeight4DataInvalid,
    IbWeightError := IbWeight4Error,
    IbWeightCalibrationInProgress := IbWeight4CalibrationInProgress,
    IbWeightSteadyState := IbWeight4SteadyState,
    IbWeightSyncError := IbWeight4SyncError,
    sNetId := '192.168.40.180.3.1' (*Adres ADS Mastera do tarowania*),
    nSlaveAddr := 1013 (*Adres wagi do tarowania*),
    iStationIndex := 35,
    sStationName := "Waga 4",
    bWarning1 := bWeight4Warning1,
    eRunningState => eWeight4RunningState,
    bError => Weight4Error.bError,
    nErrorNr => Weight4Error.nErrorCode,
    sErrorDescription => Weight4Error.sErrorString,
    sErrorDescription2 => Weight4Error.sErrorString2,
    sErrorStationName => Weight4Error.sStationName,
    udiStationID => Weight4Error.udiStationID,
    lrMeasuredWeight => VIS.lrWeight4Measured,
    lrChartWeight => lrWeight4Chart (*tylko do wykresu*),
    QbWeightStartCalibration => QbWeight4StartCalibration,
    QbWeightDisableCalibration => QbWeight4DisableCalibration,
    QbWeightInputFreeze => QbWeight4InputFreeze,
    QbWeightSampleMode => QbWeight4SampleMode,
    QbWeightTara => QbWeight4Tara); // FB_BeckhoffEL3356Weight
eWeight4State := fbWeight4.eState;

// NETWORK 2
END_ACTION

ACTION aWeight5:
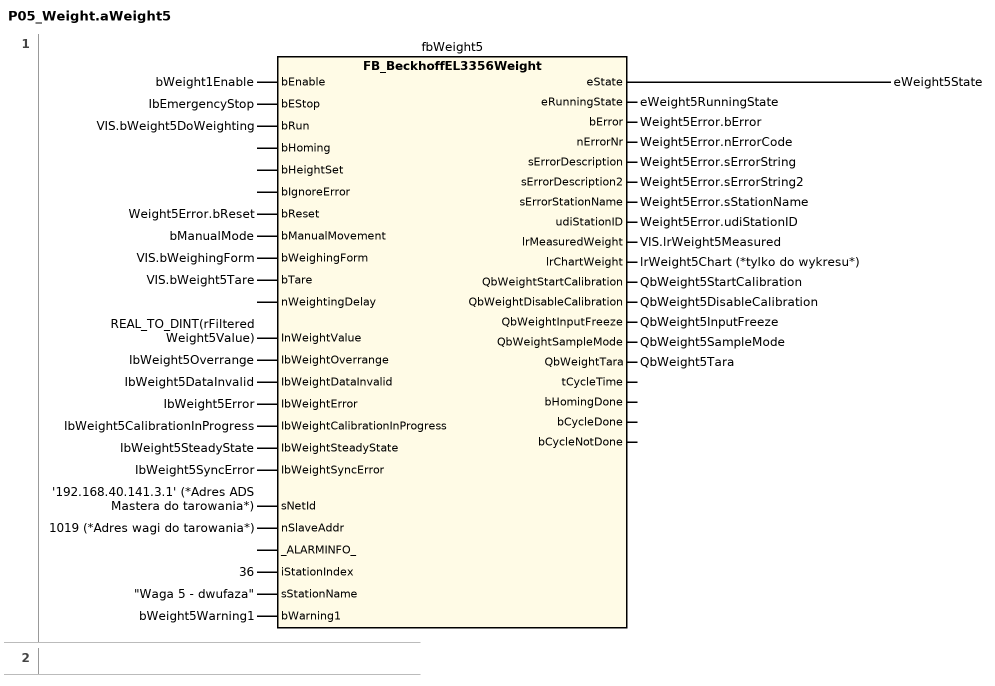
// NETWORK 1
fbWeight5(
    bEnable := bWeight1Enable,
    bEStop := IbEmergencyStop,
    bRun := VIS.bWeight5DoWeighting,
    bReset := Weight5Error.bReset,
    bManualMovement := bManualMode,
    bWeighingForm := VIS.bWeighingForm,
    bTare := VIS.bWeight5Tare,
    InWeightValue := REAL_TO_DINT(rFilteredWeight5Value),
    IbWeightOverrange := IbWeight5Overrange,
    IbWeightDataInvalid := IbWeight5DataInvalid,
    IbWeightError := IbWeight5Error,
    IbWeightCalibrationInProgress := IbWeight5CalibrationInProgress,
    IbWeightSteadyState := IbWeight5SteadyState,
    IbWeightSyncError := IbWeight5SyncError,
    sNetId := '192.168.40.141.3.1' (*Adres ADS Mastera do tarowania*),
    nSlaveAddr := 1019 (*Adres wagi do tarowania*),
    iStationIndex := 36,
    sStationName := "Waga 5 - dwufaza",
    bWarning1 := bWeight5Warning1,
    eRunningState => eWeight5RunningState,
    bError => Weight5Error.bError,
    nErrorNr => Weight5Error.nErrorCode,
    sErrorDescription => Weight5Error.sErrorString,
    sErrorDescription2 => Weight5Error.sErrorString2,
    sErrorStationName => Weight5Error.sStationName,
    udiStationID => Weight5Error.udiStationID,
    lrMeasuredWeight => VIS.lrWeight5Measured,
    lrChartWeight => lrWeight5Chart (*tylko do wykresu*),
    QbWeightStartCalibration => QbWeight5StartCalibration,
    QbWeightDisableCalibration => QbWeight5DisableCalibration,
    QbWeightInputFreeze => QbWeight5InputFreeze,
    QbWeightSampleMode => QbWeight5SampleMode,
    QbWeightTara => QbWeight5Tara); // FB_BeckhoffEL3356Weight
eWeight5State := fbWeight5.eState;

// NETWORK 2
END_ACTION

ACTION aWeight6:
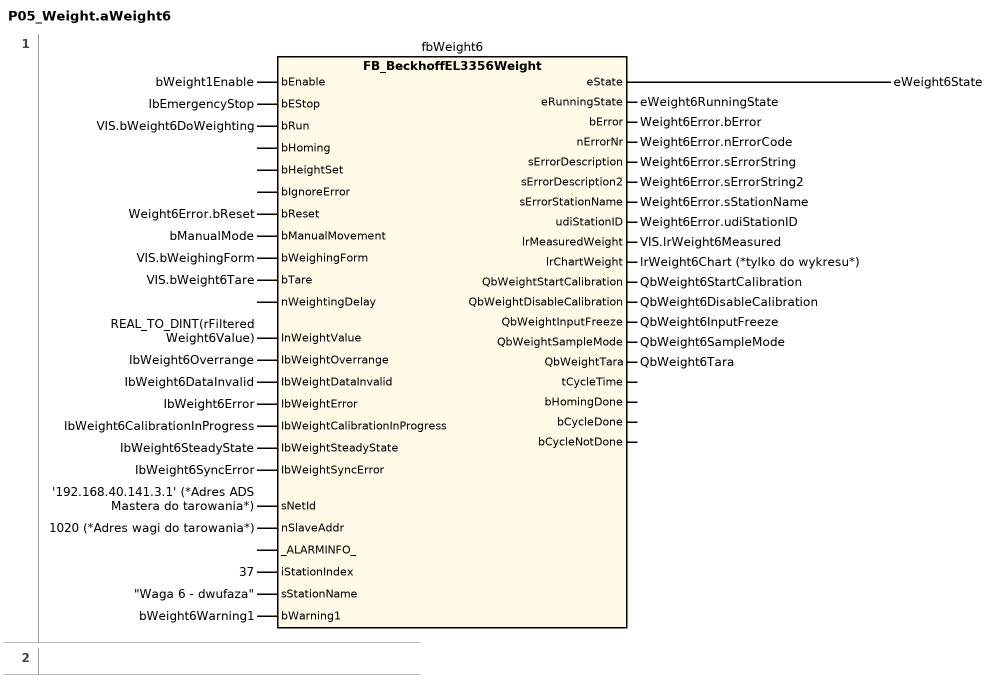
// NETWORK 1
fbWeight6(
    bEnable := bWeight1Enable,
    bEStop := IbEmergencyStop,
    bRun := VIS.bWeight6DoWeighting,
    bReset := Weight6Error.bReset,
    bManualMovement := bManualMode,
    bWeighingForm := VIS.bWeighingForm,
    bTare := VIS.bWeight6Tare,
    InWeightValue := REAL_TO_DINT(rFilteredWeight6Value),
    IbWeightOverrange := IbWeight6Overrange,
    IbWeightDataInvalid := IbWeight6DataInvalid,
    IbWeightError := IbWeight6Error,
    IbWeightCalibrationInProgress := IbWeight6CalibrationInProgress,
    IbWeightSteadyState := IbWeight6SteadyState,
    IbWeightSyncError := IbWeight6SyncError,
    sNetId := '192.168.40.141.3.1' (*Adres ADS Mastera do tarowania*),
    nSlaveAddr := 1020 (*Adres wagi do tarowania*),
    iStationIndex := 37,
    sStationName := "Waga 6 - dwufaza",
    bWarning1 := bWeight6Warning1,
    eRunningState => eWeight6RunningState,
    bError => Weight6Error.bError,
    nErrorNr => Weight6Error.nErrorCode,
    sErrorDescription => Weight6Error.sErrorString,
    sErrorDescription2 => Weight6Error.sErrorString2,
    sErrorStationName => Weight6Error.sStationName,
    udiStationID => Weight6Error.udiStationID,
    lrMeasuredWeight => VIS.lrWeight6Measured,
    lrChartWeight => lrWeight6Chart (*tylko do wykresu*),
    QbWeightStartCalibration => QbWeight6StartCalibration,
    QbWeightDisableCalibration => QbWeight6DisableCalibration,
    QbWeightInputFreeze => QbWeight6InputFreeze,
    QbWeightSampleMode => QbWeight6SampleMode,
    QbWeightTara => QbWeight6Tara); // FB_BeckhoffEL3356Weight
eWeight6State := fbWeight6.eState;

// NETWORK 2
END_ACTION

END_PROGRAM

(* stored: Version 1.1.0.1, ProductVersion 3.1.4026.13, FileIdentifier 8a4157822fb89c35ce98bb1ce9e77f230a6a6fe9, FileSignature 4a686dfead6649d319bab954d2ae9ee1c3d9d78b99341f9ae3850577fa39a58675c8ffec948732832739a5afcd9ba84a804870b5e78aeccaaed8a520a030917425abe2d0f05e2fc58c6c4af87d45a62fbf99a7cf856e58a5fc7adff76d334657134cd2229926ac9f5b70d45d55311ce33f827a9aa25009faaf47ebf435d48bdcf61fceb0ac35f3bc2e6f3ce546dbfeae4b4f47d79c2f86ef9764c9fe863cde57de3f9ad9281bbd696eb8320d1cf2805b0ab878693f81b33a0c9cf31d6ebec5279eb99c97988a98f5b021061a1dcb895485e6617f8a2a8f6a4f14aa7c9f79855729e1e4a46d3ad52240a10fb10a8bc208e807b565c74234c69c8e9b522313f7e3
   POU P05_Weight: Id {05bbbfe4-5c17-4ccc-940d-f7506e5ee82e}, SpecialFunc None
   Action ACT_WeightChartDrawers: Id {c706a3e0-fc01-42bc-9fbd-fa553e41361e}
   Action ACT_WeightStation: Id {eb03ee02-74e3-4d7f-8f39-d2ef734bed74}
   Action ACT_WeightStation2Phase: Id {d55b1c8e-c473-4c97-8f65-2f9e9603d15f}
   Action aFilter: Id {054fb911-064d-4d6b-b330-bfe3d6d0d99b}
   Action aWeight1: Id {7fc79ad1-5182-4002-a670-bdba3e2cc754}
   Action aWeight2: Id {c1e9e86f-34b5-4f96-850a-3aa0af4afad3}
   Action aWeight3: Id {e337eae0-c667-44ca-8694-1b899de79a0e}
   Action aWeight4: Id {033978de-4b31-48fe-b9cf-117d9253b757}
   Action aWeight5: Id {01b99d4d-782c-4419-bf9c-e522814b67a8}
   Action aWeight6: Id {ae8879e0-fe27-4d78-8d8c-69affe156502} *)
